TYPE ST_PumpSettings :
STRUCT
	iMeterVelocity			: UINT;
	iRunVelocity			: UINT;
	iEmptyFactor			: UINT;
	iFillolventTubesFactor	: UINT;
END_STRUCT
END_TYPE

(* stored: Version 1.1.0.1, ProductVersion 3.1.4024.12
   DUT ST_PumpSettings: Id {06bb022e-562d-4d40-8f37-3e81a50b923a} *)
